// TIA Portal V20 export
TYPE "typeEm2MonitoringUserDefine"
// stored: Access Published, Namespace Unit1
   STRUCT
      executionEnabled : Bool;
      manualControlEnabled { ExternalWritable := 'False'} : Bool;
      manualModeChangeEnabled { ExternalWritable := 'False'} : Bool;
   END_STRUCT;
END_TYPE
